FUNCTION_BLOCK FB_Auswertung
VAR_INPUT
	I_Manuel			:BOOL;	
	I_RNr				:INT;				// Reaktornummer für korrekte Zuweisung von SystemStatusWord		
	I_ControlWord		:RezeptControlWord;
	I_SystemStatusWord	:SystemStatusWord;
	I_SekCW				:SekControlWord;
END_VAR
VAR_OUTPUT
	O_StatusWord		:RezeptStatusWord; 
	O_SystemON			:BOOL;
END_VAR
VAR
	V_Status			:INT;						// Variable für Case-Switch
	V_Aktiv				:BOOL;						// Variable für Case-Management
	V_GF_Switch			:INT;						// Definiert welche GF durchgegührt werden soll	
	V_SekRe				:BOOL;						// Wird aktiviert falls Reaktor als Sekundärreaktor eingesetzt wird
	V_SekReady			:BOOL;
	V_SekActiv			:BOOL;
END_VAR

// Befindet sich System in Manuel-Modus
IF I_Manuel THEN
	V_Status := 0;
END_IF  

IF NOT I_Manuel AND NOT V_Aktiv THEN
	V_Status := 1;
END_IF

// Auswertung des SystemStatusWords 
CASE I_RNr OF 
	1:	V_SekReady := I_SystemStatusWord.R1_Ready;
		V_SekActiv := I_SystemStatusWord.R1_Activ;
	
	2:	V_SekReady := I_SystemStatusWord.R2_Ready;
		V_SekActiv := I_SystemStatusWord.R2_Activ;
	
	3:	V_SekReady := I_SystemStatusWord.R3_Ready;
		V_SekActiv := I_SystemStatusWord.R3_Activ;
	
	4:	V_SekReady := I_SystemStatusWord.R4_Ready;
		V_SekActiv := I_SystemStatusWord.R4_Activ;
		
	5:	V_SekReady := I_SystemStatusWord.R5_Ready;
		V_SekActiv := I_SystemStatusWord.R5_Activ;
	
	6:	V_SekReady := I_SystemStatusWord.R6_Ready;
		V_SekActiv := I_SystemStatusWord.R6_Activ;
	
	7:	V_SekReady := I_SystemStatusWord.R7_Ready;
		V_SekActiv := I_SystemStatusWord.R7_Activ;
END_CASE

CASE V_Status OF
	0: // System im Manuel-Modus
		
	//==================================================================================================
	1: // Auswerten von Controlwords bezüglich Systemstart
		IF I_ControlWord.PowerOn AND NOT O_SystemON THEN
			V_Aktiv := TRUE;
			V_Status := 2;
		END_IF
		
		// Auswertung von Sekundärreaktor-Controlword bezüglich Empfänger-Prozes 
		CASE I_RNr OF 
			1: V_SekRe := I_SekCW.R1;
			2: V_SekRe := I_SekCW.R2;
			3: V_SekRe := I_SekCW.R3;
			4: V_SekRe := I_SekCW.R4;
			5: V_SekRe := I_SekCW.R5;
			6: V_SekRe := I_SekCW.R6;
			7: V_SekRe := I_SekCW.R7;
		END_CASE
		
		IF V_SekRe THEN
			V_Aktiv := TRUE;
			V_Status := 2;
		END_IF
	
	//==================================================================================================
	2: // System wird eingeschaltet
			O_SystemON := TRUE;
			O_StatusWord.SysReady := TRUE;
			
			IF GVL.Bedien_Power THEN
				V_Status := 3;
			END_IF
	//==================================================================================================
	3: // Leitung wird definiert
			
			V_Status := 4;
	//==================================================================================================
	4: // Prozess wird durchgeführt
		IF I_ControlWord.Enlteermenge > 0 THEN
			V_GF_Switch := 1;
			Kommunikation.Entleeren.M_START();
			V_Status := 5;
		END_IF
		
		IF I_ControlWord.Pumpmenge > 0 THEN
			V_GF_Switch := 2;
			Kommunikation.Pumpen.M_START();
			V_Status := 5;
		END_IF
		
		IF I_ControlWord.Haltedauer > 0 THEN
			V_GF_Switch := 3;
			V_Status := 5;
		END_IF
		
		IF I_ControlWord.Ruehrdauer > 0 THEN
			V_GF_Switch := 4;
			Kommunikation.Ruehren.M_START();
			V_Status := 5;
		END_IF
		
		IF I_ControlWord.Wartedauer > 0 THEN
			V_GF_Switch := 5;
			Kommunikation.Warten.M_START();
			V_Status := 5;
		END_IF
		
		IF I_ControlWord.Zirkulierdauer > 0 THEN
			V_GF_Switch := 6;
			Kommunikation.Zirkulieren.M_START();
			V_Status := 5;
		END_IF
		
		IF V_SekRe THEN
			V_GF_Switch := 7;
			Kommunikation.Befuellen.M_START();
			V_Status := 5;
		END_IF
		
	//==================================================================================================
	5: // System wartete auf Abschluss von Prozess
		CASE V_GF_Switch OF 
			1:	ACT_GF_Entleeren();
				IF Kommunikation.Entleeren.P_Status = 0 THEN
					V_Status := 6;
				END_IF
				
			2:	ACT_GF_Pumpen();
				IF Kommunikation.Pumpen.P_Status = 0 THEN
					V_Status := 6;
				END_IF
				
			3: //
			
			4:	ACT_GF_Ruehren();
				IF Kommunikation.Ruehren.P_Status = 0 THEN
					V_Status := 6;
				END_IF
				
			5:	ACT_GF_Warten();
				IF Kommunikation.Warten.P_Status = 0 THEN
					V_Status := 6;
				END_IF
				
			6:	ACT_GF_Zirkulieren();
				IF Kommunikation.Zirkulieren.P_Status = 0 THEN
					V_Status := 6;
				END_IF
				
			7: ACT_GF_Befuellen();
				IF Kommunikation.Befuellen.P_Status = 0 THEN
					V_Status := 6;
				END_IF
		END_CASE
	//==================================================================================================
	6: // System wird ausgeschalten
		IF NOT I_ControlWord.PowerOn THEN
			O_SystemON := FALSE;
			O_StatusWord.SysReady := FALSE;
			V_Aktiv := FALSE; 
			V_Status := 1;
		END_IF
END_CASE

ACTION ACT_GF_Befuellen:
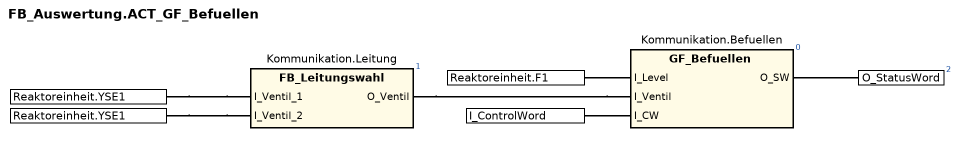
Kommunikation.Befuellen(
    I_Level := Reaktoreinheit.F1,
    I_Ventil := Kommunikation.Leitung.O_Ventil,
    I_CW := I_ControlWord); // GF_Befuellen
Kommunikation.Leitung(I_Ventil_1 := Reaktoreinheit.YSE1, I_Ventil_2 := Reaktoreinheit.YSE1); // FB_Leitungswahl
O_StatusWord := Kommunikation.Befuellen.O_SW;
END_ACTION

ACTION ACT_GF_Entleeren:
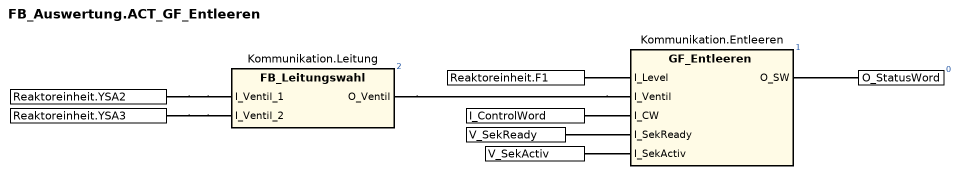
O_StatusWord := Kommunikation.Entleeren.O_SW;
Kommunikation.Entleeren(
    I_Level := Reaktoreinheit.F1,
    I_Ventil := Kommunikation.Leitung.O_Ventil,
    I_CW := I_ControlWord,
    I_SekReady := V_SekReady,
    I_SekActiv := V_SekActiv); // GF_Entleeren
Kommunikation.Leitung(I_Ventil_1 := Reaktoreinheit.YSA2, I_Ventil_2 := Reaktoreinheit.YSA3); // FB_Leitungswahl
END_ACTION

ACTION ACT_GF_Pumpen:
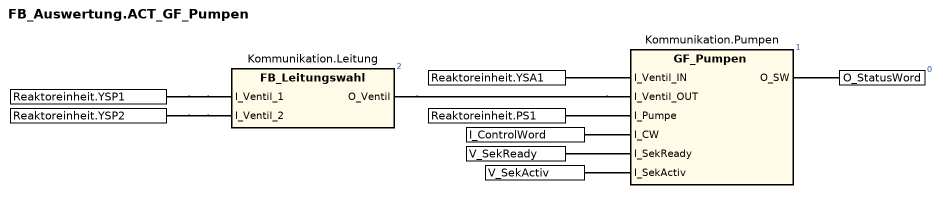
O_StatusWord := Kommunikation.Pumpen.O_SW;
Kommunikation.Pumpen(
    I_Ventil_IN := Reaktoreinheit.YSA1,
    I_Ventil_OUT := Kommunikation.Leitung.O_Ventil,
    I_Pumpe := Reaktoreinheit.PS1,
    I_CW := I_ControlWord,
    I_SekReady := V_SekReady,
    I_SekActiv := V_SekActiv); // GF_Pumpen
Kommunikation.Leitung(I_Ventil_1 := Reaktoreinheit.YSP1, I_Ventil_2 := Reaktoreinheit.YSP2); // FB_Leitungswahl
END_ACTION

ACTION ACT_GF_Ruehren:
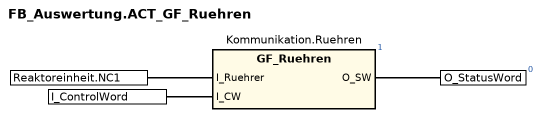
O_StatusWord := Kommunikation.Ruehren.O_SW;
Kommunikation.Ruehren(I_Ruehrer := Reaktoreinheit.NC1, I_CW := I_ControlWord); // GF_Ruehren
END_ACTION

ACTION ACT_GF_Warten:
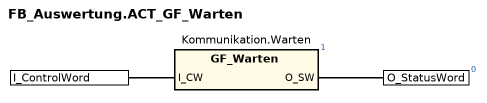
O_StatusWord := Kommunikation.Warten.O_SW;
Kommunikation.Warten(I_CW := I_ControlWord); // GF_Warten
END_ACTION

ACTION ACT_GF_Zirkulieren:
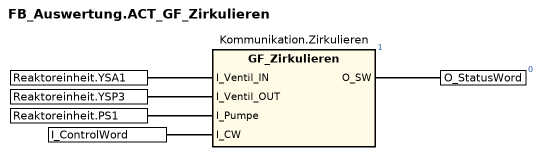
O_StatusWord := Kommunikation.Zirkulieren.O_SW;
Kommunikation.Zirkulieren(
    I_Ventil_IN := Reaktoreinheit.YSA1,
    I_Ventil_OUT := Reaktoreinheit.YSP3,
    I_Pumpe := Reaktoreinheit.PS1,
    I_CW := I_ControlWord); // GF_Zirkulieren
END_ACTION

END_FUNCTION_BLOCK

(* stored: Version 1.1.0.1, ProductVersion 3.1.4024.12
   POU FB_Auswertung: Id {c05caf1a-4e85-4b15-b759-42af766126d1}, SpecialFunc None
   Action ACT_GF_Befuellen: Id {d7245a94-2b35-4d27-a17e-5a30739f3f68}
   Action ACT_GF_Entleeren: Id {fe72f81c-be04-4b50-a27a-4d648bc8c63c}
   Action ACT_GF_Pumpen: Id {658c8ff4-9f1e-4d92-a42e-2f4328264cd7}
   Action ACT_GF_Ruehren: Id {9001b75e-4bfa-42e1-8d8a-3b08a12675a6}
   Action ACT_GF_Warten: Id {ed3b8586-88c5-476e-b06c-94cc6435962e}
   Action ACT_GF_Zirkulieren: Id {4e867aee-05f8-49e9-9b7d-19cacf114c3f} *)
